// TIA Portal V19 export
DATA_BLOCK "HmiInterface"   // DB152
// stored: MemoryReserve 100, Namespace Unit.Em0
   VAR
      em : "LAF_typeEmInterface";
   END_VAR
BEGIN
END_DATA_BLOCK
